(* IEC 61131-3 sources: trust-platform/examples/plant_demo/src, 4 files *)

(* ---- types.st ---- *)
TYPE
    E_PumpState : (Idle := 0, Starting := 1, Running := 2, Fault := 3);

    ST_PumpCommand :
    STRUCT
        Enable : BOOL;
        TargetSpeed : REAL;
    END_STRUCT;

    ST_PumpStatus :
    STRUCT
        Running : BOOL;
        State : E_PumpState;
        ActualSpeed : REAL;
        Alarm : UDINT;
    END_STRUCT;
END_TYPE

(* ---- fb_pump.st ---- *)
FUNCTION_BLOCK FB_Pump
VAR_INPUT
    Command : ST_PumpCommand;
END_VAR
VAR_OUTPUT
    Status : ST_PumpStatus;
END_VAR
VAR
    ramp_timer : TON;
    ramp : REAL;
END_VAR
VAR CONSTANT
    RAMP_TIME : TIME := T#1s;
END_VAR

Status.Running := FALSE;
Status.Alarm := 0;

IF NOT Command.Enable THEN
    Status.State := E_PumpState#Idle;
    Status.ActualSpeed := 0.0;
    ramp := 0.0;
    ramp_timer(IN := FALSE);
ELSE
    CASE Status.State OF
        E_PumpState#Idle:
            Status.State := E_PumpState#Starting;
            ramp_timer(IN := TRUE, PT := RAMP_TIME);
        E_PumpState#Starting:
            ramp_timer(IN := TRUE, PT := RAMP_TIME);
            IF ramp_timer.Q THEN
                Status.State := E_PumpState#Running;
            ELSE
                ramp := ramp + 0.2;
            END_IF
        E_PumpState#Running:
            Status.Running := TRUE;
            ramp := Command.TargetSpeed;
        E_PumpState#Fault:
            Status.Running := FALSE;
            Status.Alarm := 16#BEEF;
    END_CASE
END_IF

Status.ActualSpeed := ramp;
END_FUNCTION_BLOCK

(* ---- config.st ---- *)
CONFIGURATION PlantDemo
TASK Fast (INTERVAL := T#100ms, PRIORITY := 1);
PROGRAM P1 WITH Fast : PlantProgram;
VAR_CONFIG
    P1.StartCmd AT %IX0.0 : BOOL;
    P1.SpeedRaw AT %IW0 : INT;
    P1.HaltReq AT %QX0.0 : BOOL;
END_VAR
END_CONFIGURATION

(* ---- program.st ---- *)
PROGRAM PlantProgram
VAR
    Pump : FB_Pump;
    Cmd : ST_PumpCommand;
    Status : ST_PumpStatus;
    StartCmd : BOOL;
    SpeedRaw : INT;
    SpeedSet : REAL;
    HaltReq : BOOL;
END_VAR

Cmd.Enable := StartCmd AND NOT HaltReq;
SpeedSet := INT_TO_REAL(SpeedRaw);
Cmd.TargetSpeed := SpeedSet;

Pump(Command := Cmd);
Status := Pump.Status;
HaltReq := FALSE;
IF Status.State = E_PumpState#Fault THEN
    HaltReq := TRUE;
END_IF
END_PROGRAM
